TYPE ST_System_AFA_Stellwert :
STRUCT
	Anford_Pumpe			: BOOL;
	Anford_Pumpe_760        : BOOL;
	Anford_Regelventil		: BOOL;
	Anford_Regelventil_Ost	: BOOL;
	Anford_Regelventil_West	: BOOL;
	Einschaltperiode_Max	: TIME := T#10S;
	Einschalten				: BOOL;
	Temp_Vorl				: REAL;
END_STRUCT
END_TYPE

(* stored: Version 1.1.0.1, ProductVersion 3.1.4024.9
   DUT ST_System_AFA_Stellwert: Id {0bd4a6f0-4203-4857-a330-541cffd56681} *)
